(* IEC 61131-3 sources: repolevel_ST_code_completion/extract_code/轴控/FB105_轴控制集/FB50_虚轴控制, 4 files *)

(* ---- A01_轴控主块.st ---- *)
PROGRAM A01_轴控主块
VAR
	FB_AxisControl_AxisVirtual : FB_轴控块;
	FB_AxisStop_AxisVirtual : FB_轴停止触发块;
	SMC_ChangeGearingRatio0 : SMC_ChangeGearingRatio;
END_VAR

VAR_INPUT
END_VAR

VAR_OUTPUT
END_VAR

VAR_IN_OUT
END_VAR

FB_AxisControl_AxisVirtual(
    (* =============== 输入参数 ( := ) =============== *)
    Enable             := ,                        (* 图中未连接，留空 *)
    JogFor             := bAxisVirtual_JogFor,
    JogBack            := bAxisVirtual_JogBack,
    JogVelocity        := rAxisVirtual_JogVelSet,   (* JogVelocity 连线到 rAxisVirtual_JogVelSet *)
    StopExecute        := bAxisVirtual_StopExcute,
    ResetExecute       := HMI_b复位,                (* ResetExecute 连线到 HMI_b复位 *)

    AbsExecute         := ,                        (* 图中未连接，留空 *)
    AbsPosition        := rAxisVirtual_AbsPositionSet,
    AbsVelocity        := rAxisVirtual_AbsVelSet,
    AbsAcceleration    := ,                        (* 图中未连接，留空 *)
    AbsDeceleration    := ,                        (* 图中未连接，留空 *)

    RelExecute         := ,                        (* 图中未连接，留空 *)
    RelPosition        := rAxisVirtual_RelPositionSet,
    RelVelocity        := rAxisVirtual_RelVelSet,
    RelAcceleration    := ,                        (* 图中未连接，留空 *)
    RelDeceleration    := ,                        (* 图中未连接，留空 *)

    VelExecute         := ,                        (* 图中未连接，留空 *)
    VelVelocity        := rAxisVirtual_VelVelSet,

    InchForward        := ,                        (* 图中未连接，留空 *)
    InchBackward       := ,                        (* 图中未连接，留空 *)
    InchDistance       := rAxisVirtual_InchPositionSet,
    InchVelocity       := rAxisVirtual_InchVelSet,
    InchAcceleration   := ,                        (* 图中未连接，留空 *)
    InchDeceleration   := ,                        (* 图中未连接，留空 *)

    SetPosExecute      := ,                        (* 图中未连接，留空 *)
    ReStartSlaveEx     := ,                        (* 图中未连接，留空 *)
    AxisName           := AxisVirtual,              (* AxisName 连线到 AxisVirtual *)

    (* =============== 输出参数 ( => ) =============== *)
    EnableStatus       => bAxisVirtual_EnableOK,
    StopDone           => bAxisVirtual_StopDone,
    AbsDone            => bAxisVirtual_AbsDone,
    RelDone            => bAxisVirtual_RelDone,
    VelBusy            => bAxisVirtual_VelBusy,
    InchBusy           => bAxisVirtual_InchBusy,
    AxisStandstill     => bAxisVirtual_Standstill,
    AbsBusy            => bAxisVirtual_AbsBusy,
    RelBusy            => bAxisVirtual_RelBusy,
    AxisError          => bAxisVirtual_AxisError,
    AxisAccing         => bAxisVirtual_Accing,
    AxisDecing         => bAxisVirtual_Decing,
    FBErrorOccurred    => ,                        (* 图中未连接，留空 *)
    Homing             => ,                        (* 图中未连接，留空 *)
    Stopping           => ,                        (* 图中未连接，留空 *)
    ErrorID            => ,                        (* 图中未连接，留空 *)
    SetPosDone         => ,                        (* 图中未连接，留空 *)
    bOperational       => ,                        (* 图中未连接，留空 *)
	eComState          => ,
    wComState          => ,                        (* 图中未连接，留空 *)
    JogBusy            => bAxisVirtual_JogBusy      (* JogBusy 连线到 bAxisVirtual_JogBusy *)
	ReStartSlaveDone   =>
);

FB_AxisStop_AxisVirtual(
	StopExcute := bAxisVirtual_StopExcute
);

SMC_ClearFBError(
	EN := FBErrorOccured,
	pDrive := ADR(AxisVirtual),
	ENO => ,
	SMC_ClearFBError =>
);

SMC_ChangeGearingRatio0(
    (* =============== 输入参数 ( := ) =============== *)
    Axis                 := AxisVirtual,
    bExecute             := ,                            (* FBD中 bExecute 引脚未连接，留空 *)
    dwRatioTechUnitsDenom:= AxisVirtual.dwRatioTechUnitsDenom, (* 分母：连接到轴变量的 Denom *)
    iRatioTechUnitsNum   := REAL_TO_INT(HMI_rAxisVirtual_Lead), (* 分子：HMI输入的REAL转INT后连接 *)
    fPositionPeriod      := ,                            (* FBD中 fPositionPeriod 未连接，留空 *)
    iMovementType        := SMC_MOVEMENTTYPE.linear,      (* 运动类型常量连接 *)

    (* =============== 输出参数 ( => ) =============== *)
    bDone                => ,
    bBusy                => ,
    bError               => ,
    nErrorID             =>
);

AxisVirtual.iRestNumerator = 0;

(* ---- A02_数据运算.st ---- *)
(*基本速度，位置*)
rAxisVirtual_JogVelSet:=HMI_rAxisVirtual_ManualVel;

rAxisVirtual_AbsVelSet:=HMI_rAxisVirtual_AutoVel;
rAxisVirtual_RelVelSet:=HMI_rAxisVirtual_AutoVel;
rAxisVirtual_VelVelSet:=HMI_rAxisVirtual_AutoVel;
rAxisVirtual_InchVelSet:=HMI_rAxisVirtual_AutoVel;

HMI_rAxisVirtual_ActPos:=LREAL_TO_REAL(AxisVirtual.fActPosition);
HMI_rAxisVirtual_ActVel:=LREAL_TO_REAL(AxisVirtual.fActVelocity);

FB_AxisControl_AxisVirtual.AbsAcceleration:=rAxisVirtual_AbsVelSet*10000;
FB_AxisControl_AxisVirtual.AbsDeceleration:=rAxisVirtual_AbsVelSet*10000;

FB_AxisControl_AxisVirtual.RelAcceleration:=rAxisVirtual_RelVelSet*10000;
FB_AxisControl_AxisVirtual.RelDeceleration:=rAxisVirtual_RelVelSet*10000;

FB_AxisControl_AxisVirtual.InchAcceleration:=rAxisVirtual_InchVelSet*10000;
FB_AxisControl_AxisVirtual.InchDeceleration:=rAxisVirtual_InchVelSet*10000;

(*正负限位*)
IF bAxisVirtual_LimitEnable AND bAxisVirtual_HomeDone THEN
	AxisVirtual.bSWLimitEnable:=TRUE;
	AxisVirtual.fSWLimitPositive:=HMI_rAxisVirtual_LimitPostive;
	AxisVirtual.fSWLimitNegative:=HMI_rAxisVirtual_LimitNegative;
	AxisVirtual.fSWLimitDeceleration:=1000000;
	ELSE
	AxisVirtual.bSWLimitEnable:=FALSE;
END_IF

(* ---- A03_原点回归.st ---- *)
PROGRAM A03_原点回归
VAR
    MC_SetPosition_0 : SM3_Basic.MC_SetPosition; (* 声明位置设置功能块 *)
END_VAR

VAR_INPUT
END_VAR

VAR_OUTPUT
END_VAR

VAR_IN_OUT
END_VAR

(* 调用MC_SetPosition功能块，实现轴位置设置 *)
MC_SetPosition_0(
    Axis := AxisVirtual,
    Execute := ,
    Position := 0,
    Mode := 0,
    Done => ,
    Busy => ,
    Error => ,
    ErrorID =>
);

(* ---- FB50_虚轴控制.st ---- *)
PROGRAM FB50_虚轴控制
VAR
	FB_AxisMotionDiag_AxisVirtual: FB_轴通讯状态块;
	SMC_SetControllerMode0: SMC_SetControllerMode;
	SMC_SetTorque0: SMC_SetTorque;
	SMC_ChangeGearingRatio0: SMC_ChangeGearingRatio;
    MC_SetPosition_0: SM3_Basic.MC_SetPosition;
	MC_GearIn_0: SM3_Basic.MC_GearIn;
	MC_GearOut_0: SM3_Basic.MC_GearOut;
	FB_AxisStop_AxisVirtual: FB_轴停止触发块;

	fb_CommunicationOK: TON;
END_VAR

(*轴通讯状态*)
bAxisVirtual_CommunicationOK:=FB_AxisMotionDiag_AxisVirtual.EtherCATBusOK;

FB_AxisMotionDiag_AxisVirtual(Axis_bCommunication:= AxisVirtual.bCommunication,
                        Axis_wCommunicationState:= AxisVirtual.wCommunicationState,
                        EtherCATBusOK=> );

fb_CommunicationOK(IN:= bAxisVirtual_CommunicationOK, PT:= T#3S, Q=> , ET=> );

(*轴使能操作*)
IF NOT HMI_bAxisVirtual_PowerOff AND fb_CommunicationOK.Q THEN
	FB_AxisControl_AxisVirtual.Enable:=TRUE;
	ELSE
	FB_AxisControl_AxisVirtual.Enable:=FALSE;
END_IF

(*轴控点动*)
IF HMI_bAxisVirtual_JogForward AND bAxisVirtual_EnableOK AND NOT bAxisVirtual_Error AND b非急停手动模式 AND NOT bAxisVirtual_JogBack THEN
	bAxisVirtual_JogFor:=TRUE;
	ELSE
	bAxisVirtual_JogFor:=FALSE;
END_IF
IF HMI_bAxisVirtual_BackForward AND bAxisVirtual_EnableOK AND NOT bAxisVirtual_Error AND b非急停手动模式 AND NOT bAxisVirtual_JogFor THEN
	bAxisVirtual_JogBack:=TRUE;
	ELSE
	bAxisVirtual_JogBack:=FALSE;
END_IF

(*轴控寸动*)
IF bAxisVirtual_InchForExcute AND bAxisVirtual_EnableOK AND NOT bAxisVirtual_Error AND NOT FB_AxisControl_AxisVirtual.InchBackward THEN
	FB_AxisControl_AxisVirtual.InchForward:=TRUE;
	ELSE
	FB_AxisControl_AxisVirtual.InchForward:=FALSE;
END_IF
IF bAxisVirtual_InchBackExcute AND bAxisVirtual_EnableOK AND NOT bAxisVirtual_Error AND NOT FB_AxisControl_AxisVirtual.InchForward THEN
	FB_AxisControl_AxisVirtual.InchBackward:=TRUE;
	ELSE
	FB_AxisControl_AxisVirtual.InchBackward:=FALSE;
END_IF

(*轴控绝对运动*)
IF bAxisVirtual_AbsExcute AND bAxisVirtual_EnableOK AND NOT bAxisVirtual_Error THEN
	FB_AxisControl_AxisVirtual.AbsExcute:=TRUE;
	ELSE
	FB_AxisControl_AxisVirtual.AbsExcute:=FALSE;
END_IF

(*轴控相对运动*)
IF bAxisVirtual_RelExcute AND bAxisVirtual_EnableOK AND NOT bAxisVirtual_Error THEN
	FB_AxisControl_AxisVirtual.RelExcute:=TRUE;
	ELSE
	FB_AxisControl_AxisVirtual.RelExcute:=FALSE;
END_IF
